{attribute 'GeneratedUsingTerminal: EL5001-0000-1016'}
{attribute addProperty BoxType "EL5001-0000-1016"}
{attribute addProperty Id "StatusAT %I*USINT1ValueAT %I*UDINT4"}
{attribute addProperty CRC "3710677834"}
{attribute addProperty Size "5"}
TYPE Channel_DD2C734A :
STRUCT
	{attribute addProperty Name "Status"}
	Status AT %I* : USINT;
	{attribute addProperty Name "Value"}
	Value AT %I* : UDINT;
END_STRUCT
END_TYPE

(* stored: Version 1.2.0.0, ProductVersion 3.1.4024.9
   DUT Channel_DD2C734A: Id {998dcb79-c093-42d8-b44c-9d462903fed7} *)
